// TIA Portal V16 export
// export: Created 2021-06-18T09:03:48.924053Z, ExportSetting WithDefaults, DisplayName Totally Integrated Automation Portal, DisplayVersion V16 Update 2, DisplayName TIA Portal Version Control Interface, DisplayVersion V16 Update 2, DisplayName TIA Portal Openness, DisplayVersion V16 Update 2, DisplayName TIA Portal Teamcenter Gateway, DisplayVersion V16, DisplayName SINAMICS Startdrive Advanced, DisplayVersion V16, DisplayName SINAMICS Startdrive G130, G150, S120, S150, SINAMICS MV, S210, DisplayVersion V16, DisplayName SINAMICS Startdrive G110M, G120, G120C, G120D, G120P, DisplayVersion V16, DisplayName STEP 7 Professional, DisplayVersion V16 Update 2, DisplayName STEP 7 Safety, DisplayVersion V16, DisplayName WinCC Advanced, DisplayVersion V16 Update 2
VAR_GLOBAL   // PLC tag table "Default tag table"
   Tag_1 AT %M1.1 : Bool;
   Tag_2 AT %M1.2 : Bool;
   Tag_3 AT %M666.5 : Bool;
   Tag_4 AT %MB444 : Byte;
   Tag_5 AT %M4.4 : Bool;
   Tag_6 AT %Q2.4 : Bool;
END_VAR
